FUNCTION_BLOCK FB_Clutch
VAR_INPUT
	Lh_in:BOOL; (*Left hand clutch in switch*)
	Lh_out:BOOL; (*Left hand clutch out switch*)
	Rh_in:BOOL; (*Right hand clutch in switch*)
	Rh_out:BOOL; (*Right hand clutch out switch*)
	Lh_movement:BOOL; (*Movement on left hand drum*)
	Rh_movement:BOOL; (*Movement on right hand drum*)
	Lh_raw_depth:DINT; (*Left conveyance raw depth*)
	Rh_raw_depth:DINT; (*Right conveyance raw depth*)
	Allowed_travel_when_out:DINT; (*Amount of travel allowed while engaging/disengaging a clutch*)
END_VAR
VAR_OUTPUT
	tr_Lh_in_and_out:BOOL; (*Left hand clutch in and out switches both energised*)
	tr_Rh_in_and_out:BOOL; (*Right hand clutch in and out switches both energised*)
	tr_Lh_out_movement:BOOL; (*Movement was detected on the left hand drum when the left clutch was out*)
	tr_Rh_out_movement:BOOL; (*Movement was detected on the right hand drum when the right clutch was out*)
	tr_Lh_not_in_movement:BOOL; (*Movement was detected on the left hand drum when the left clutch was not in*)
	tr_Rh_not_in_movement:BOOL; (*Movement was detected on the right hand drum when the right clutch was not in*)
	cs_Too_much_travel_clutching:BOOL; (*There was too much drum travel while engaging/disengaging a clutch*)
	hmi_Status:WORD; (*Status bits for HMI*)
END_VAR
VAR
	TON_0: TON;
	TON_1: TON;
	TON_2: TON;
	TON_3: TON;
	Lh_start_depth: DINT;
	RS_0: RS;
	Rh_start_depth: DINT;
	RS_1: RS;
END_VAR

M_Clutch_data();
M_Clutch_faults();
M_Too_much_travel();

METHOD M_Clutch_data
VAR_INPUT
END_VAR

VAR
	BIT_TO_WORD_V0_0: FB_BIT_TO_WORD_V0;
END_VAR
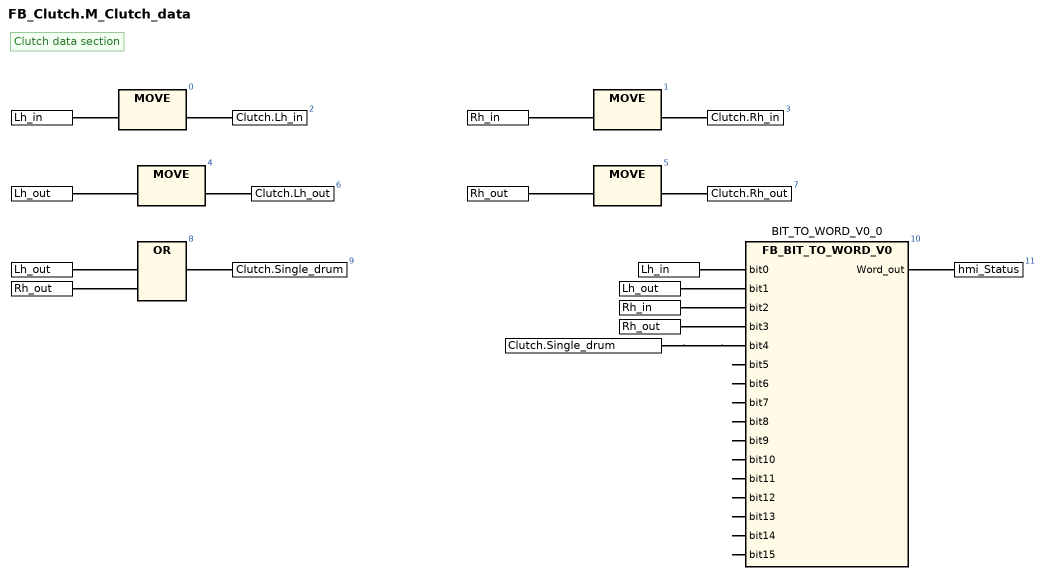
// Clutch data section
Clutch.Lh_in := Lh_in;
Clutch.Rh_in := Rh_in;
Clutch.Lh_out := Lh_out;
Clutch.Rh_out := Rh_out;
Clutch.Single_drum := Lh_out OR Rh_out;
BIT_TO_WORD_V0_0(bit0 := Lh_in, bit1 := Lh_out, bit2 := Rh_in, bit3 := Rh_out, bit4 := Clutch.Single_drum); // FB_BIT_TO_WORD_V0
hmi_Status := BIT_TO_WORD_V0_0.Word_out;
END_METHOD

METHOD M_Clutch_faults
VAR_INPUT
END_VAR
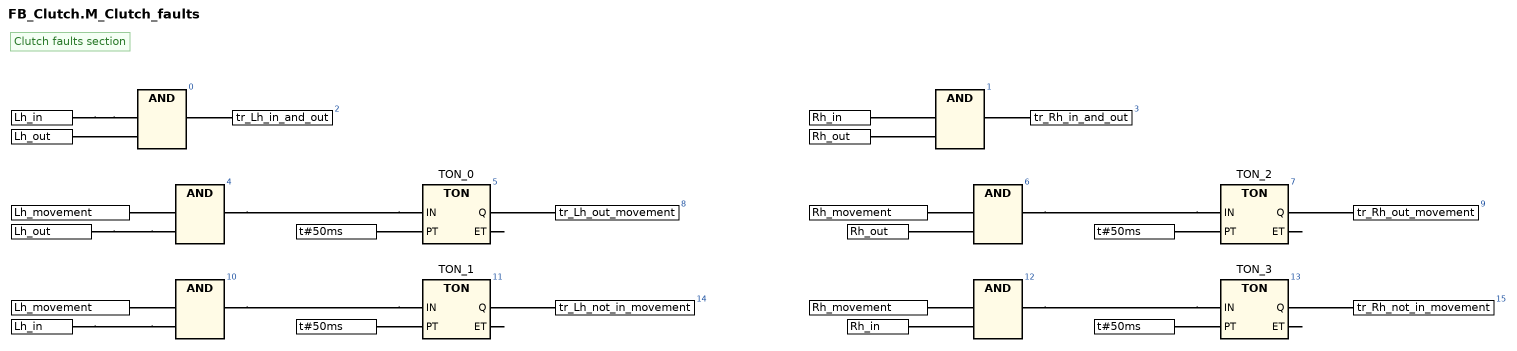
// Clutch faults section
tr_Lh_in_and_out := Lh_in AND Lh_out;
tr_Rh_in_and_out := Rh_in AND Rh_out;
TON_0(IN := Lh_movement AND Lh_out, PT := t#50ms); // TON
TON_2(IN := Rh_movement AND Rh_out, PT := t#50ms); // TON
tr_Lh_out_movement := TON_0.Q;
tr_Rh_out_movement := TON_2.Q;
TON_1(IN := Lh_movement AND Lh_in, PT := t#50ms); // TON
TON_3(IN := Rh_movement AND Rh_in, PT := t#50ms); // TON
tr_Lh_not_in_movement := TON_1.Q;
tr_Rh_not_in_movement := TON_3.Q;
END_METHOD

METHOD M_Too_much_travel
VAR_INPUT
END_VAR
VAR_INST // added by the converter: edge detectors and wires of the graphical bodies
    _w1, _w3 : ANY;
    _w2, _w4 : DINT;
END_VAR
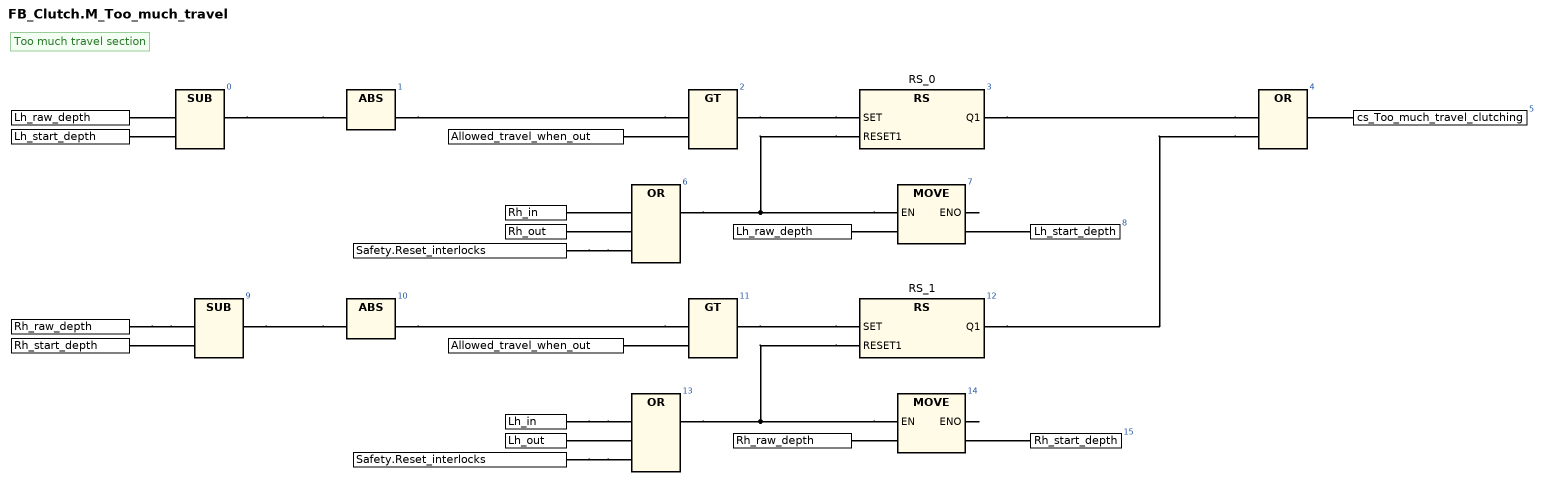
// Too much travel section
RS_0(SET := ABS(Lh_raw_depth - Lh_start_depth) > Allowed_travel_when_out, RESET1 := _w1); // RS
cs_Too_much_travel_clutching := RS_0.Q1 OR RS_1.Q1;
_w1 := Rh_in OR Rh_out OR Safety.Reset_interlocks;
IF _w1 THEN _w2 := Lh_raw_depth; END_IF
Lh_start_depth := _w2;
RS_1(SET := ABS(Rh_raw_depth - Rh_start_depth) > Allowed_travel_when_out, RESET1 := _w3); // RS
_w3 := Lh_in OR Lh_out OR Safety.Reset_interlocks;
IF _w3 THEN _w4 := Rh_raw_depth; END_IF
Rh_start_depth := _w4;
END_METHOD

END_FUNCTION_BLOCK

(* stored: Version 1.1.0.1, ProductVersion 3.1.4024.0
   POU FB_Clutch: Id {b7a093e0-243f-430e-afed-272cb59f6ae8}, SpecialFunc None
   Method M_Clutch_data: Id {fbc9329b-cdb5-41d3-be6d-4e780531c171}
   Method M_Clutch_faults: Id {3012f220-18ae-4f9f-8169-363c8fff1f4a}
   Method M_Too_much_travel: Id {6e6efc1e-b899-4739-9f3a-95f717dbd697} *)
